// Mitsubishi GX Developer project: 壓碗機_20130207   PLC: FX1N

PROGRAM MAIN
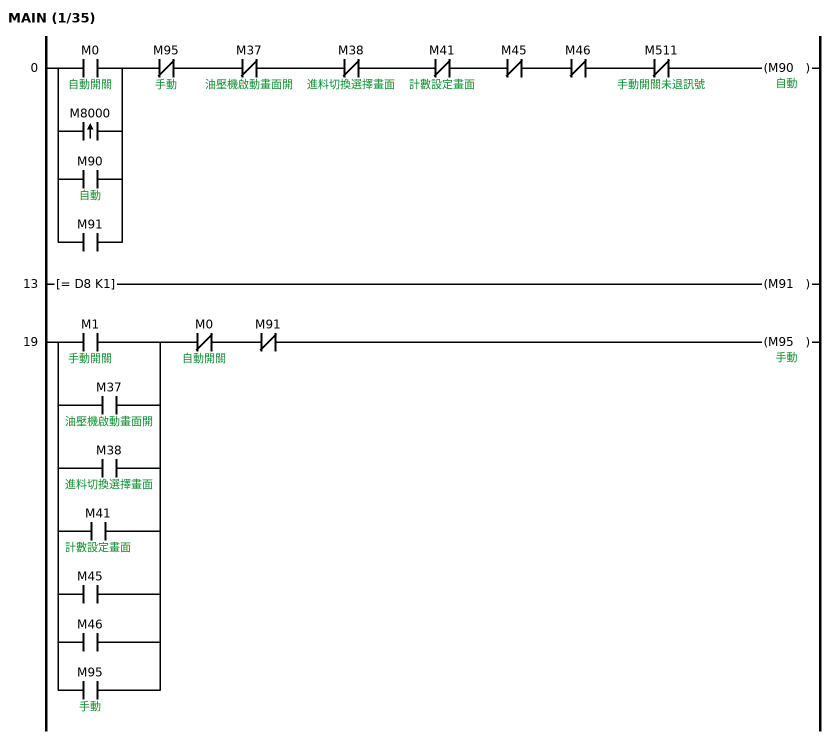
0     LD      M0  ; 自動開關
      ORP     M8000
      OR      M90  ; 自動
      OR      M91
      ANI     M95  ; 手動
      ANI     M37  ; 油壓機啟動畫面開
      ANI     M38  ; 進料切換選擇畫面
      ANI     M41  ; 計數設定畫面
      ANI     M45
      ANI     M46
      ANI     M511  ; 手動開關未退訊號
      OUT     M90  ; 自動
13    LD=     D8 K1
      OUT     M91
19    LD      M1  ; 手動開關
      OR      M37  ; 油壓機啟動畫面開
      OR      M38  ; 進料切換選擇畫面
      OR      M41  ; 計數設定畫面
      OR      M45
      OR      M46
      OR      M95  ; 手動
      ANI     M0  ; 自動開關
      ANI     M91
      OUT     M95  ; 手動
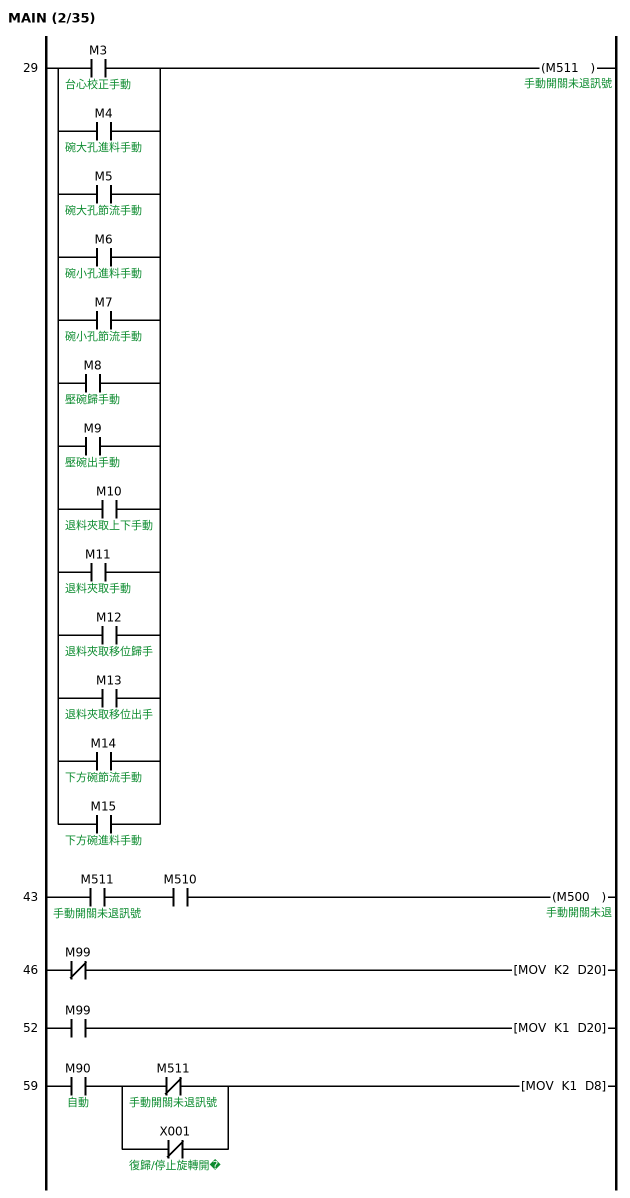
29    LD      M3  ; 台心校正手動
      OR      M4  ; 碗大孔進料手動
      OR      M5  ; 碗大孔節流手動
      OR      M6  ; 碗小孔進料手動
      OR      M7  ; 碗小孔節流手動
      OR      M8  ; 壓碗歸手動
      OR      M9  ; 壓碗出手動
      OR      M10  ; 退料夾取上下手動
      OR      M11  ; 退料夾取手動
      OR      M12  ; 退料夾取移位歸手
      OR      M13  ; 退料夾取移位出手
      OR      M14  ; 下方碗節流手動
      OR      M15  ; 下方碗進料手動
      OUT     M511  ; 手動開關未退訊號
43    LD      M511  ; 手動開關未退訊號
      AND     M510
      OUT     M500  ; 手動開關未退
46    LDI     M99
      MOV     K2 D20
52    LD      M99
      MOV     K1 D20
59    LD      M90  ; 自動
      LDI     M511  ; 手動開關未退訊號
      ORI     X001  ; 復歸/停止旋轉開�
      ANB
      MOV     K1 D8
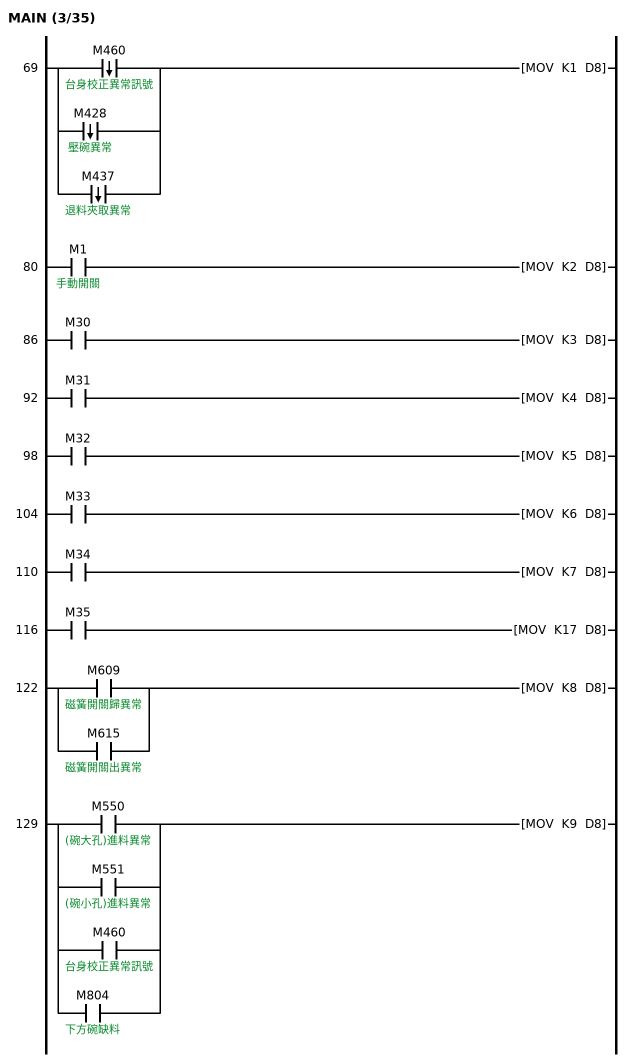
69    LDF     M460  ; 台身校正異常訊號
      ORF     M428  ; 壓碗異常
      ORF     M437  ; 退料夾取異常
      MOV     K1 D8
80    LD      M1  ; 手動開關
      MOV     K2 D8
86    LD      M30
      MOV     K3 D8
92    LD      M31
      MOV     K4 D8
98    LD      M32
      MOV     K5 D8
104   LD      M33
      MOV     K6 D8
110   LD      M34
      MOV     K7 D8
116   LD      M35
      MOV     K17 D8
122   LD      M609  ; 磁簧開關歸異常
      OR      M615  ; 磁簧開關出異常
      MOV     K8 D8
129   LD      M550  ; (碗大孔)進料異常
      OR      M551  ; (碗小孔)進料異常
      OR      M460  ; 台身校正異常訊號
      OR      M804  ; 下方碗缺料
      MOV     K9 D8
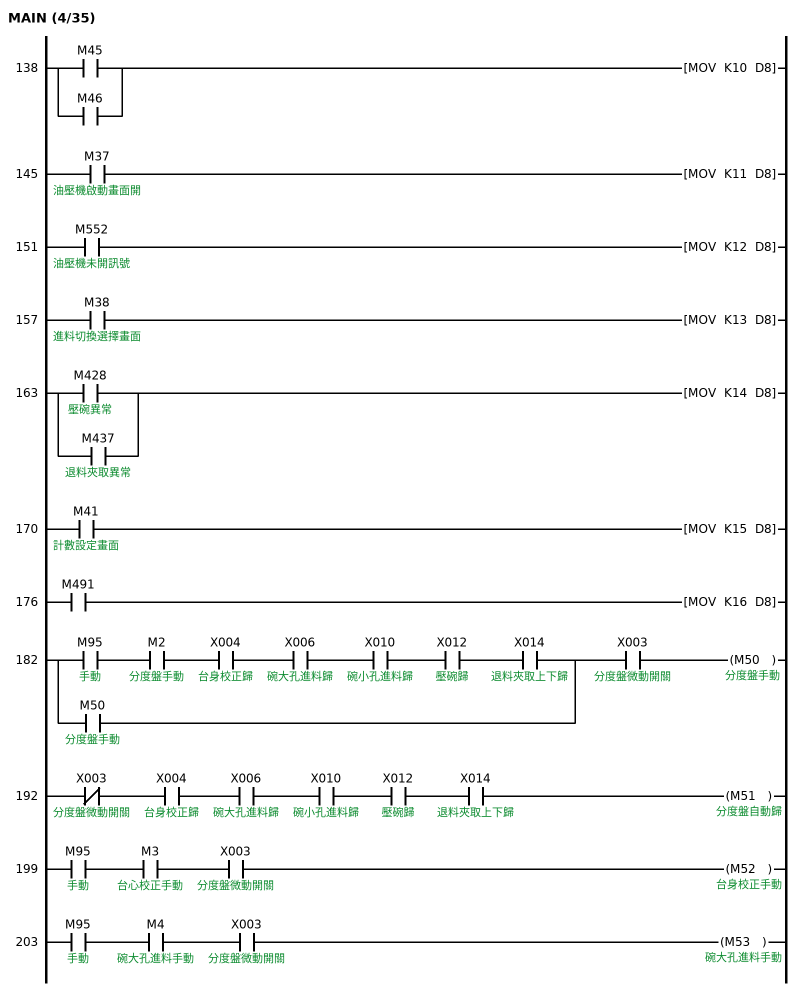
138   LD      M45
      OR      M46
      MOV     K10 D8
145   LD      M37  ; 油壓機啟動畫面開
      MOV     K11 D8
151   LD      M552  ; 油壓機未開訊號
      MOV     K12 D8
157   LD      M38  ; 進料切換選擇畫面
      MOV     K13 D8
163   LD      M428  ; 壓碗異常
      OR      M437  ; 退料夾取異常
      MOV     K14 D8
170   LD      M41  ; 計數設定畫面
      MOV     K15 D8
176   LD      M491
      MOV     K16 D8
182   LD      M95  ; 手動
      AND     M2  ; 分度盤手動
      AND     X004  ; 台身校正歸
      AND     X006  ; 碗大孔進料歸
      AND     X010  ; 碗小孔進料歸
      AND     X012  ; 壓碗歸
      AND     X014  ; 退料夾取上下歸
      OR      M50  ; 分度盤手動
      AND     X003  ; 分度盤微動開關
      OUT     M50  ; 分度盤手動
192   LDI     X003  ; 分度盤微動開關
      AND     X004  ; 台身校正歸
      AND     X006  ; 碗大孔進料歸
      AND     X010  ; 碗小孔進料歸
      AND     X012  ; 壓碗歸
      AND     X014  ; 退料夾取上下歸
      OUT     M51  ; 分度盤自動歸
199   LD      M95  ; 手動
      AND     M3  ; 台心校正手動
      AND     X003  ; 分度盤微動開關
      OUT     M52  ; 台身校正手動
203   LD      M95  ; 手動
      AND     M4  ; 碗大孔進料手動
      AND     X003  ; 分度盤微動開關
      OUT     M53  ; 碗大孔進料手動
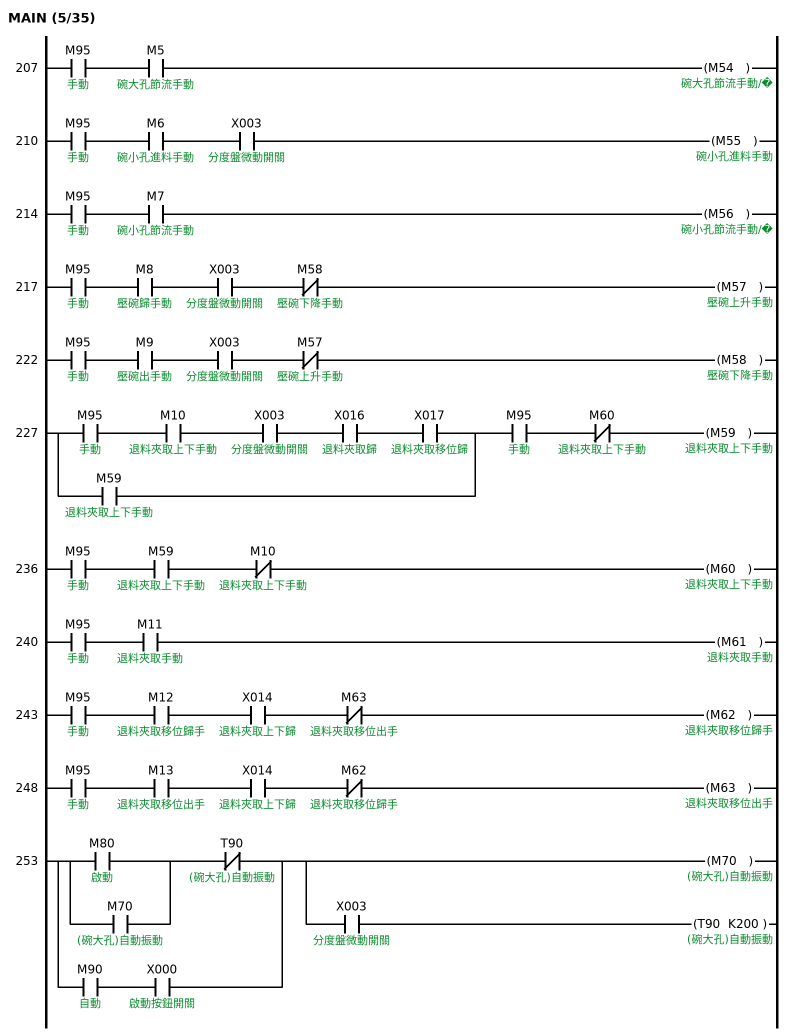
207   LD      M95  ; 手動
      AND     M5  ; 碗大孔節流手動
      OUT     M54  ; 碗大孔節流手動/�
210   LD      M95  ; 手動
      AND     M6  ; 碗小孔進料手動
      AND     X003  ; 分度盤微動開關
      OUT     M55  ; 碗小孔進料手動
214   LD      M95  ; 手動
      AND     M7  ; 碗小孔節流手動
      OUT     M56  ; 碗小孔節流手動/�
217   LD      M95  ; 手動
      AND     M8  ; 壓碗歸手動
      AND     X003  ; 分度盤微動開關
      ANI     M58  ; 壓碗下降手動
      OUT     M57  ; 壓碗上升手動
222   LD      M95  ; 手動
      AND     M9  ; 壓碗出手動
      AND     X003  ; 分度盤微動開關
      ANI     M57  ; 壓碗上升手動
      OUT     M58  ; 壓碗下降手動
227   LD      M95  ; 手動
      AND     M10  ; 退料夾取上下手動
      AND     X003  ; 分度盤微動開關
      AND     X016  ; 退料夾取歸
      AND     X017  ; 退料夾取移位歸
      OR      M59  ; 退料夾取上下手動
      AND     M95  ; 手動
      ANI     M60  ; 退料夾取上下手動
      OUT     M59  ; 退料夾取上下手動
236   LD      M95  ; 手動
      AND     M59  ; 退料夾取上下手動
      ANI     M10  ; 退料夾取上下手動
      OUT     M60  ; 退料夾取上下手動
240   LD      M95  ; 手動
      AND     M11  ; 退料夾取手動
      OUT     M61  ; 退料夾取手動
243   LD      M95  ; 手動
      AND     M12  ; 退料夾取移位歸手
      AND     X014  ; 退料夾取上下歸
      ANI     M63  ; 退料夾取移位出手
      OUT     M62  ; 退料夾取移位歸手
248   LD      M95  ; 手動
      AND     M13  ; 退料夾取移位出手
      AND     X014  ; 退料夾取上下歸
      ANI     M62  ; 退料夾取移位歸手
      OUT     M63  ; 退料夾取移位出手
253   LD      M80  ; 啟動
      OR      M70  ; (碗大孔)自動振動
      ANI     T90  ; (碗大孔)自動振動
      LD      M90  ; 自動
      AND     X000  ; 啟動按鈕開關
      ORB
      OUT     M70  ; (碗大孔)自動振動
      AND     X003  ; 分度盤微動開關
      OUT     T90 K200  ; (碗大孔)自動振動
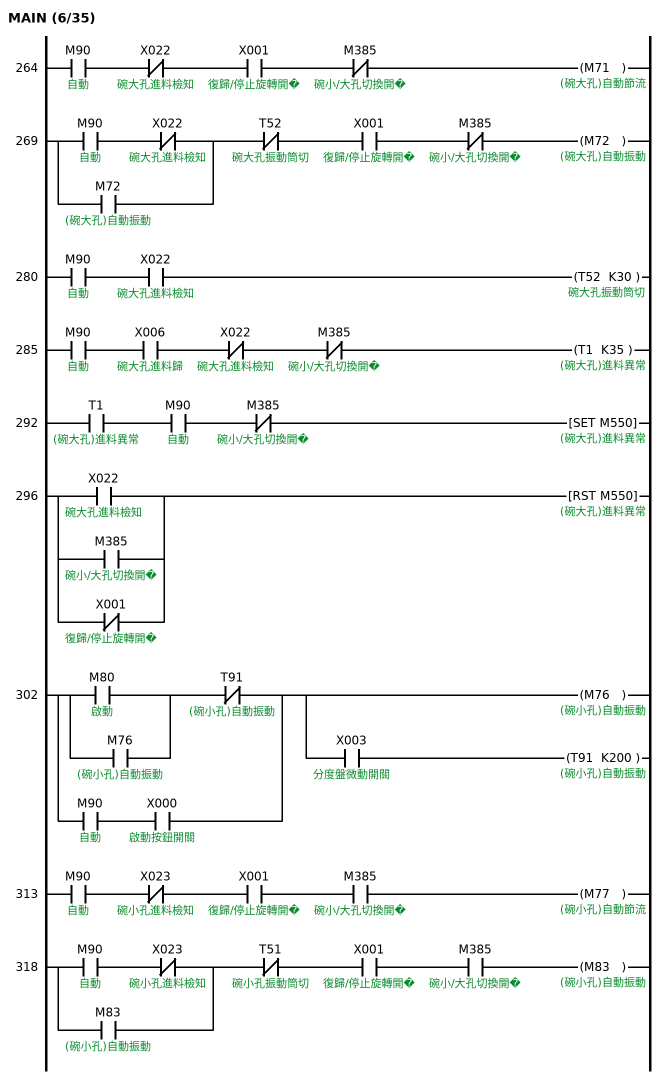
264   LD      M90  ; 自動
      ANI     X022  ; 碗大孔進料檢知
      AND     X001  ; 復歸/停止旋轉開�
      ANI     M385  ; 碗小/大孔切換開�
      OUT     M71  ; (碗大孔)自動節流
269   LD      M90  ; 自動
      ANI     X022  ; 碗大孔進料檢知
      OR      M72  ; (碗大孔)自動振動
      ANI     T52  ; 碗大孔振動筒切
      AND     X001  ; 復歸/停止旋轉開�
      ANI     M385  ; 碗小/大孔切換開�
      OUT     M72  ; (碗大孔)自動振動
280   LD      M90  ; 自動
      AND     X022  ; 碗大孔進料檢知
      OUT     T52 K30  ; 碗大孔振動筒切
285   LD      M90  ; 自動
      AND     X006  ; 碗大孔進料歸
      ANI     X022  ; 碗大孔進料檢知
      ANI     M385  ; 碗小/大孔切換開�
      OUT     T1 K35  ; (碗大孔)進料異常
292   LD      T1  ; (碗大孔)進料異常
      AND     M90  ; 自動
      ANI     M385  ; 碗小/大孔切換開�
      SET     M550  ; (碗大孔)進料異常
296   LD      X022  ; 碗大孔進料檢知
      OR      M385  ; 碗小/大孔切換開�
      ORI     X001  ; 復歸/停止旋轉開�
      RST     M550  ; (碗大孔)進料異常
302   LD      M80  ; 啟動
      OR      M76  ; (碗小孔)自動振動
      ANI     T91  ; (碗小孔)自動振動
      LD      M90  ; 自動
      AND     X000  ; 啟動按鈕開關
      ORB
      OUT     M76  ; (碗小孔)自動振動
      AND     X003  ; 分度盤微動開關
      OUT     T91 K200  ; (碗小孔)自動振動
313   LD      M90  ; 自動
      ANI     X023  ; 碗小孔進料檢知
      AND     X001  ; 復歸/停止旋轉開�
      AND     M385  ; 碗小/大孔切換開�
      OUT     M77  ; (碗小孔)自動節流
318   LD      M90  ; 自動
      ANI     X023  ; 碗小孔進料檢知
      OR      M83  ; (碗小孔)自動振動
      ANI     T51  ; 碗小孔振動筒切
      AND     X001  ; 復歸/停止旋轉開�
      AND     M385  ; 碗小/大孔切換開�
      OUT     M83  ; (碗小孔)自動振動
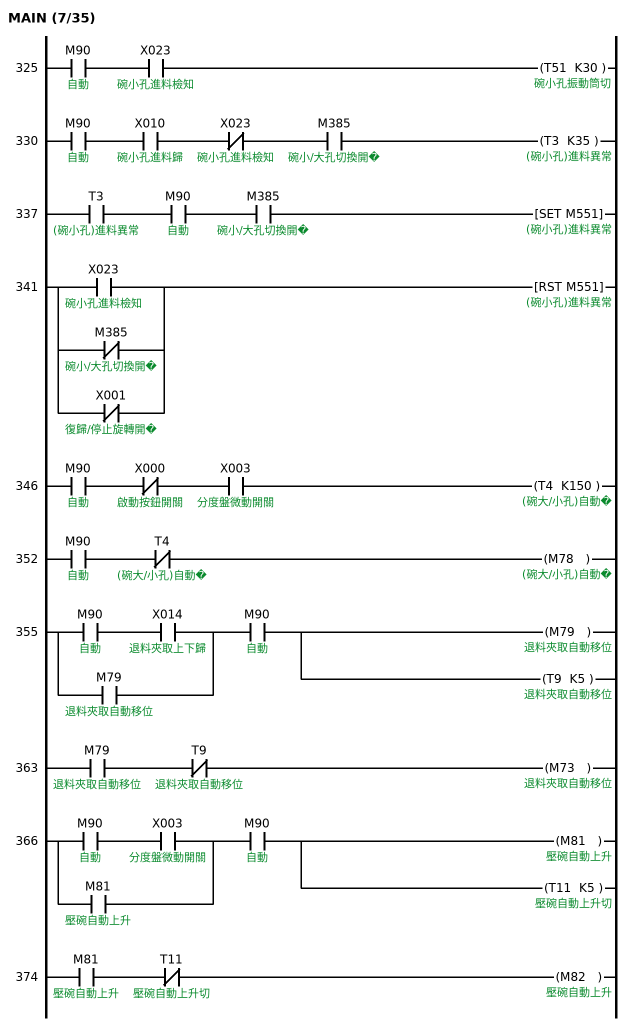
325   LD      M90  ; 自動
      AND     X023  ; 碗小孔進料檢知
      OUT     T51 K30  ; 碗小孔振動筒切
330   LD      M90  ; 自動
      AND     X010  ; 碗小孔進料歸
      ANI     X023  ; 碗小孔進料檢知
      AND     M385  ; 碗小/大孔切換開�
      OUT     T3 K35  ; (碗小孔)進料異常
337   LD      T3  ; (碗小孔)進料異常
      AND     M90  ; 自動
      AND     M385  ; 碗小/大孔切換開�
      SET     M551  ; (碗小孔)進料異常
341   LD      X023  ; 碗小孔進料檢知
      ORI     M385  ; 碗小/大孔切換開�
      ORI     X001  ; 復歸/停止旋轉開�
      RST     M551  ; (碗小孔)進料異常
346   LD      M90  ; 自動
      ANI     X000  ; 啟動按鈕開關
      AND     X003  ; 分度盤微動開關
      OUT     T4 K150  ; (碗大/小孔)自動�
352   LD      M90  ; 自動
      ANI     T4  ; (碗大/小孔)自動�
      OUT     M78  ; (碗大/小孔)自動�
355   LD      M90  ; 自動
      AND     X014  ; 退料夾取上下歸
      OR      M79  ; 退料夾取自動移位
      AND     M90  ; 自動
      OUT     M79  ; 退料夾取自動移位
      OUT     T9 K5  ; 退料夾取自動移位
363   LD      M79  ; 退料夾取自動移位
      ANI     T9  ; 退料夾取自動移位
      OUT     M73  ; 退料夾取自動移位
366   LD      M90  ; 自動
      AND     X003  ; 分度盤微動開關
      OR      M81  ; 壓碗自動上升
      AND     M90  ; 自動
      OUT     M81  ; 壓碗自動上升
      OUT     T11 K5  ; 壓碗自動上升切
374   LD      M81  ; 壓碗自動上升
      ANI     T11  ; 壓碗自動上升切
      OUT     M82  ; 壓碗自動上升
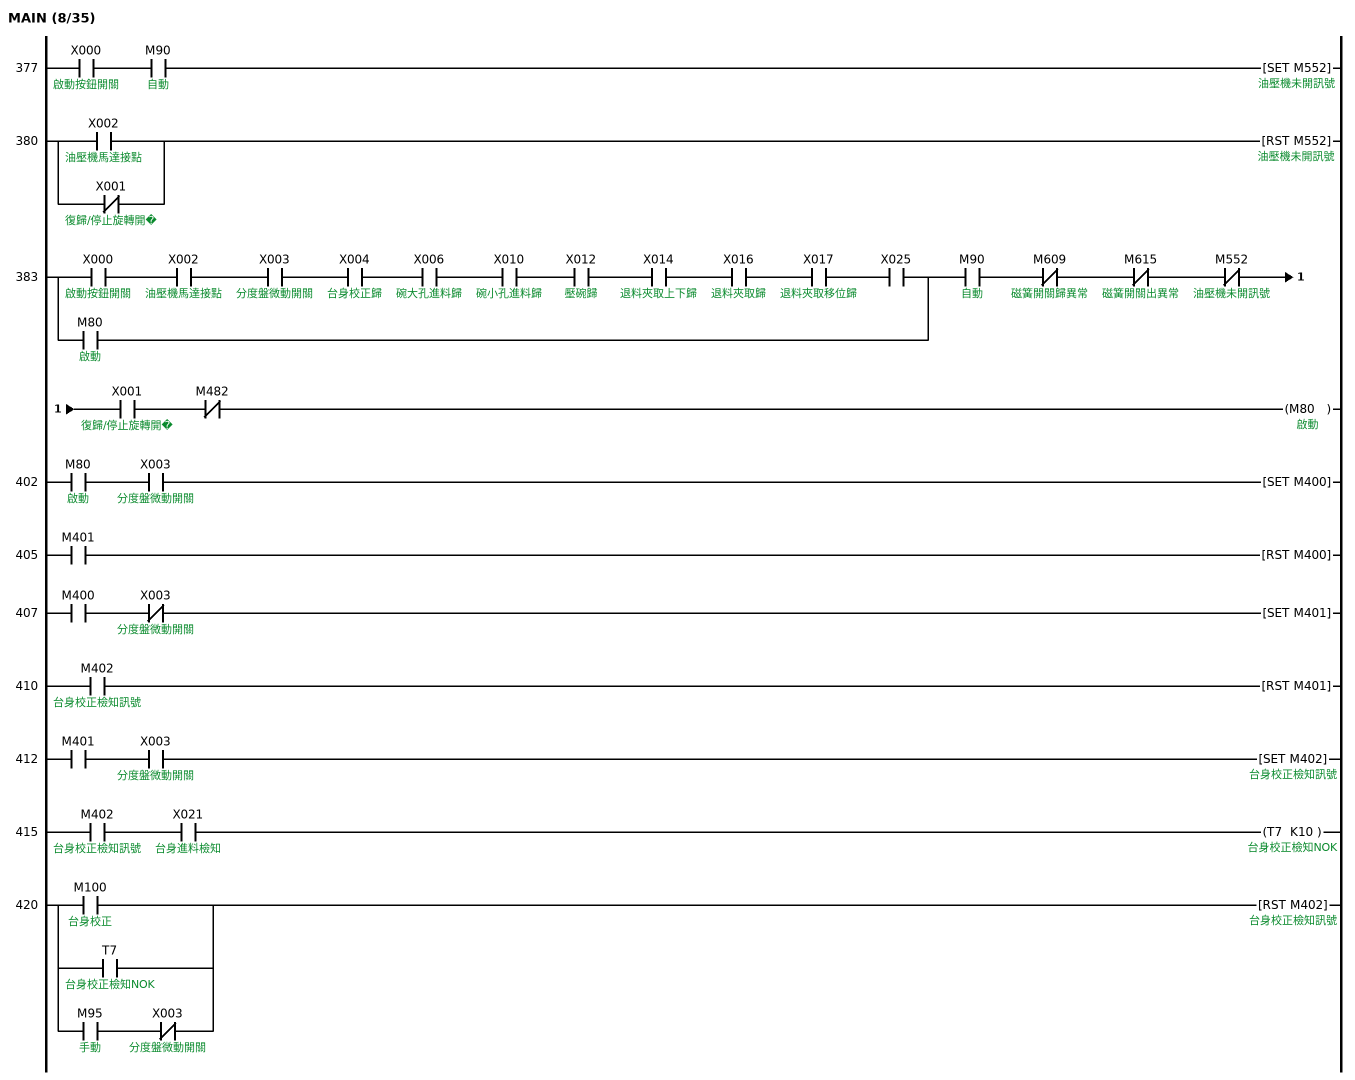
377   LD      X000  ; 啟動按鈕開關
      AND     M90  ; 自動
      SET     M552  ; 油壓機未開訊號
380   LD      X002  ; 油壓機馬達接點
      ORI     X001  ; 復歸/停止旋轉開�
      RST     M552  ; 油壓機未開訊號
383   LD      X000  ; 啟動按鈕開關
      AND     X002  ; 油壓機馬達接點
      AND     X003  ; 分度盤微動開關
      AND     X004  ; 台身校正歸
      AND     X006  ; 碗大孔進料歸
      AND     X010  ; 碗小孔進料歸
      AND     X012  ; 壓碗歸
      AND     X014  ; 退料夾取上下歸
      AND     X016  ; 退料夾取歸
      AND     X017  ; 退料夾取移位歸
      AND     X025
      OR      M80  ; 啟動
      AND     M90  ; 自動
      ANI     M609  ; 磁簧開關歸異常
      ANI     M615  ; 磁簧開關出異常
      ANI     M552  ; 油壓機未開訊號
      AND     X001  ; 復歸/停止旋轉開�
      ANI     M482
      OUT     M80  ; 啟動
402   LD      M80  ; 啟動
      AND     X003  ; 分度盤微動開關
      SET     M400
405   LD      M401
      RST     M400
407   LD      M400
      ANI     X003  ; 分度盤微動開關
      SET     M401
410   LD      M402  ; 台身校正檢知訊號
      RST     M401
412   LD      M401
      AND     X003  ; 分度盤微動開關
      SET     M402  ; 台身校正檢知訊號
415   LD      M402  ; 台身校正檢知訊號
      AND     X021  ; 台身進料檢知
      OUT     T7 K10  ; 台身校正檢知NOK
420   LD      M100  ; 台身校正
      OR      T7  ; 台身校正檢知NOK
      LD      M95  ; 手動
      ANI     X003  ; 分度盤微動開關
      ORB
      RST     M402  ; 台身校正檢知訊號
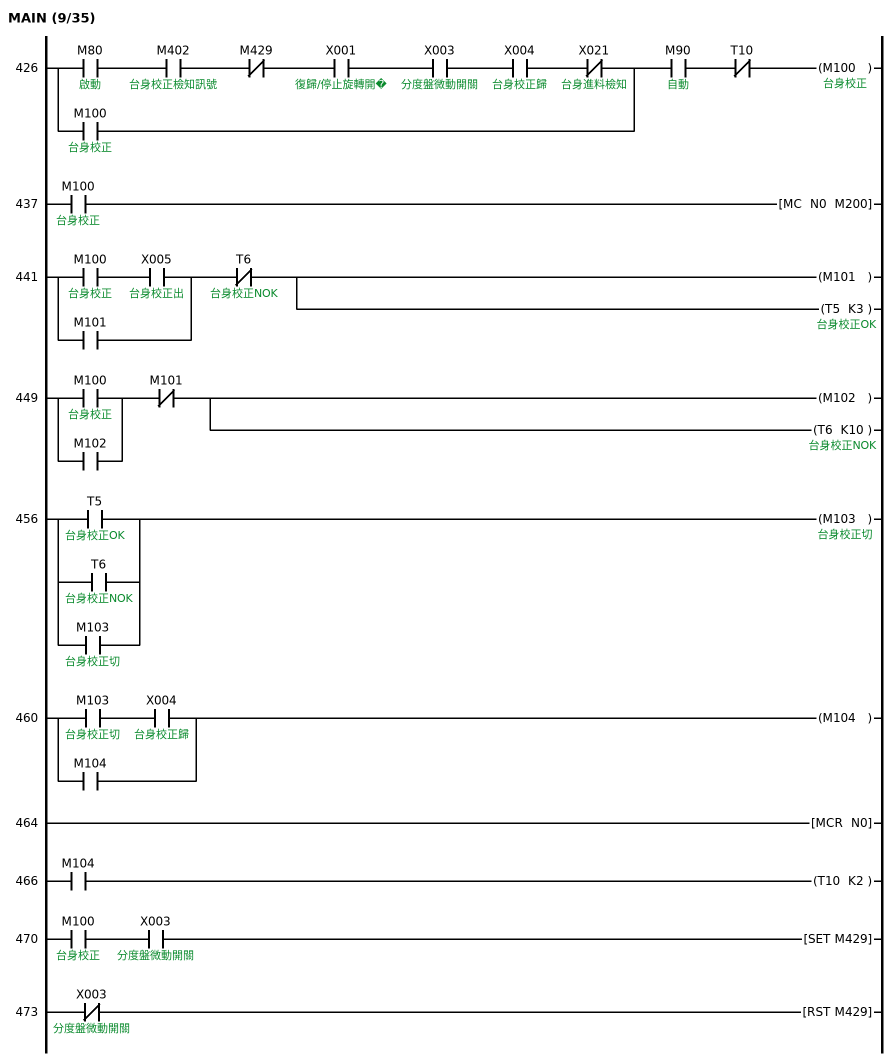
426   LD      M80  ; 啟動
      AND     M402  ; 台身校正檢知訊號
      ANI     M429
      AND     X001  ; 復歸/停止旋轉開�
      AND     X003  ; 分度盤微動開關
      AND     X004  ; 台身校正歸
      ANI     X021  ; 台身進料檢知
      OR      M100  ; 台身校正
      AND     M90  ; 自動
      ANI     T10
      OUT     M100  ; 台身校正
437   LD      M100  ; 台身校正
      MC      N0 M200
441   LD      M100  ; 台身校正
      AND     X005  ; 台身校正出
      OR      M101
      ANI     T6  ; 台身校正NOK
      OUT     M101
      OUT     T5 K3  ; 台身校正OK
449   LD      M100  ; 台身校正
      OR      M102
      ANI     M101
      OUT     M102
      OUT     T6 K10  ; 台身校正NOK
456   LD      T5  ; 台身校正OK
      OR      T6  ; 台身校正NOK
      OR      M103  ; 台身校正切
      OUT     M103  ; 台身校正切
460   LD      M103  ; 台身校正切
      AND     X004  ; 台身校正歸
      OR      M104
      OUT     M104
464   MCR     N0
466   LD      M104
      OUT     T10 K2
470   LD      M100  ; 台身校正
      AND     X003  ; 分度盤微動開關
      SET     M429
473   LDI     X003  ; 分度盤微動開關
      RST     M429
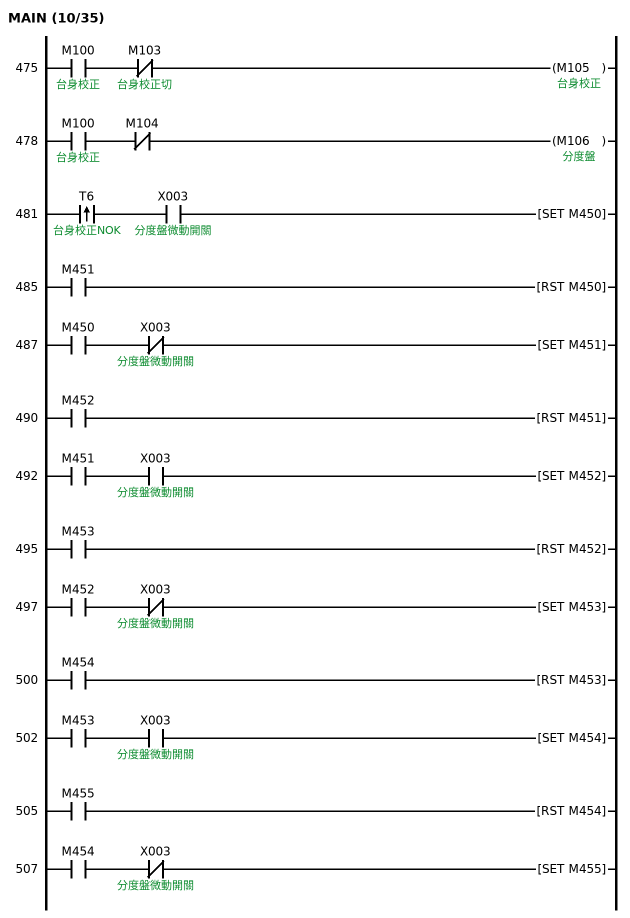
475   LD      M100  ; 台身校正
      ANI     M103  ; 台身校正切
      OUT     M105  ; 台身校正
478   LD      M100  ; 台身校正
      ANI     M104
      OUT     M106  ; 分度盤
481   LDP     T6  ; 台身校正NOK
      AND     X003  ; 分度盤微動開關
      SET     M450
485   LD      M451
      RST     M450
487   LD      M450
      ANI     X003  ; 分度盤微動開關
      SET     M451
490   LD      M452
      RST     M451
492   LD      M451
      AND     X003  ; 分度盤微動開關
      SET     M452
495   LD      M453
      RST     M452
497   LD      M452
      ANI     X003  ; 分度盤微動開關
      SET     M453
500   LD      M454
      RST     M453
502   LD      M453
      AND     X003  ; 分度盤微動開關
      SET     M454
505   LD      M455
      RST     M454
507   LD      M454
      ANI     X003  ; 分度盤微動開關
      SET     M455
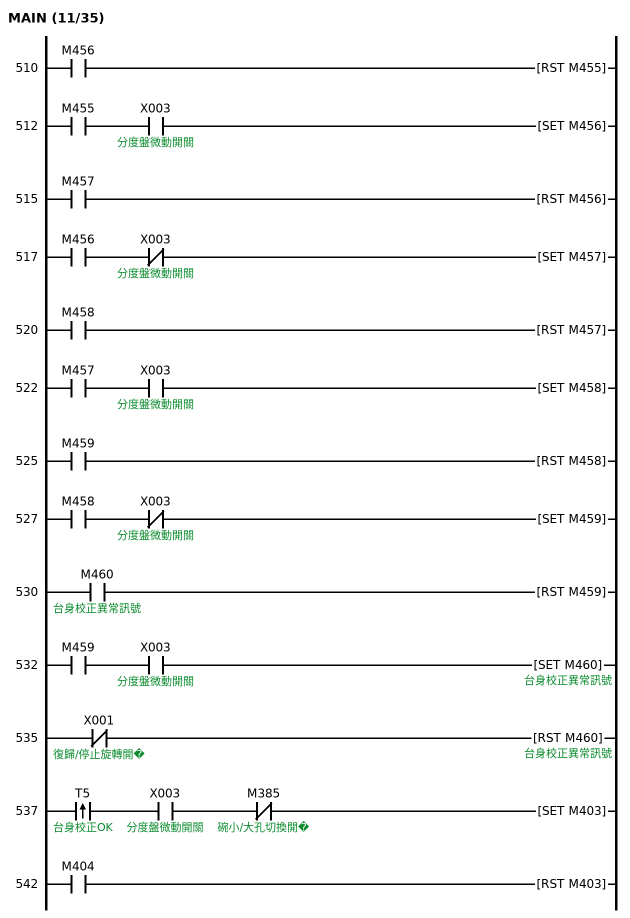
510   LD      M456
      RST     M455
512   LD      M455
      AND     X003  ; 分度盤微動開關
      SET     M456
515   LD      M457
      RST     M456
517   LD      M456
      ANI     X003  ; 分度盤微動開關
      SET     M457
520   LD      M458
      RST     M457
522   LD      M457
      AND     X003  ; 分度盤微動開關
      SET     M458
525   LD      M459
      RST     M458
527   LD      M458
      ANI     X003  ; 分度盤微動開關
      SET     M459
530   LD      M460  ; 台身校正異常訊號
      RST     M459
532   LD      M459
      AND     X003  ; 分度盤微動開關
      SET     M460  ; 台身校正異常訊號
535   LDI     X001  ; 復歸/停止旋轉開�
      RST     M460  ; 台身校正異常訊號
537   LDP     T5  ; 台身校正OK
      AND     X003  ; 分度盤微動開關
      ANI     M385  ; 碗小/大孔切換開�
      SET     M403
542   LD      M404
      RST     M403
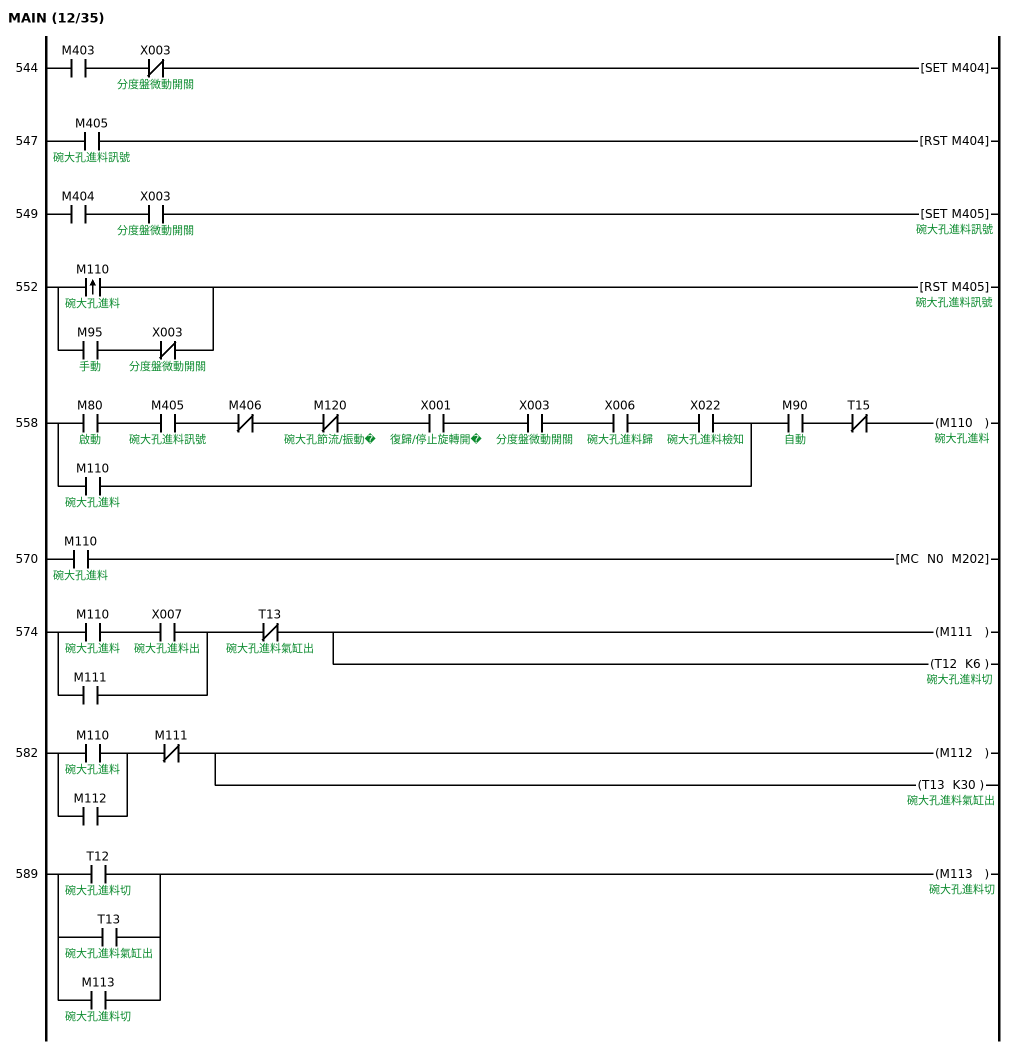
544   LD      M403
      ANI     X003  ; 分度盤微動開關
      SET     M404
547   LD      M405  ; 碗大孔進料訊號
      RST     M404
549   LD      M404
      AND     X003  ; 分度盤微動開關
      SET     M405  ; 碗大孔進料訊號
552   LDP     M110  ; 碗大孔進料
      LD      M95  ; 手動
      ANI     X003  ; 分度盤微動開關
      ORB
      RST     M405  ; 碗大孔進料訊號
558   LD      M80  ; 啟動
      AND     M405  ; 碗大孔進料訊號
      ANI     M406
      ANI     M120  ; 碗大孔節流/振動�
      AND     X001  ; 復歸/停止旋轉開�
      AND     X003  ; 分度盤微動開關
      AND     X006  ; 碗大孔進料歸
      AND     X022  ; 碗大孔進料檢知
      OR      M110  ; 碗大孔進料
      AND     M90  ; 自動
      ANI     T15
      OUT     M110  ; 碗大孔進料
570   LD      M110  ; 碗大孔進料
      MC      N0 M202
574   LD      M110  ; 碗大孔進料
      AND     X007  ; 碗大孔進料出
      OR      M111
      ANI     T13  ; 碗大孔進料氣缸出
      OUT     M111
      OUT     T12 K6  ; 碗大孔進料切
582   LD      M110  ; 碗大孔進料
      OR      M112
      ANI     M111
      OUT     M112
      OUT     T13 K30  ; 碗大孔進料氣缸出
589   LD      T12  ; 碗大孔進料切
      OR      T13  ; 碗大孔進料氣缸出
      OR      M113  ; 碗大孔進料切
      OUT     M113  ; 碗大孔進料切
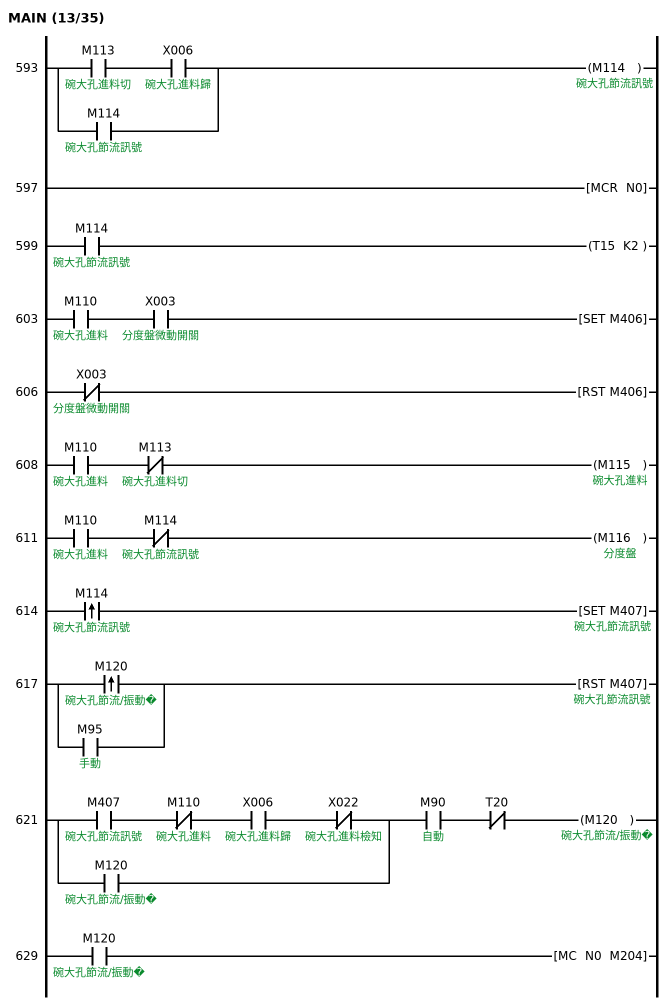
593   LD      M113  ; 碗大孔進料切
      AND     X006  ; 碗大孔進料歸
      OR      M114  ; 碗大孔節流訊號
      OUT     M114  ; 碗大孔節流訊號
597   MCR     N0
599   LD      M114  ; 碗大孔節流訊號
      OUT     T15 K2
603   LD      M110  ; 碗大孔進料
      AND     X003  ; 分度盤微動開關
      SET     M406
606   LDI     X003  ; 分度盤微動開關
      RST     M406
608   LD      M110  ; 碗大孔進料
      ANI     M113  ; 碗大孔進料切
      OUT     M115  ; 碗大孔進料
611   LD      M110  ; 碗大孔進料
      ANI     M114  ; 碗大孔節流訊號
      OUT     M116  ; 分度盤
614   LDP     M114  ; 碗大孔節流訊號
      SET     M407  ; 碗大孔節流訊號
617   LDP     M120  ; 碗大孔節流/振動�
      OR      M95  ; 手動
      RST     M407  ; 碗大孔節流訊號
621   LD      M407  ; 碗大孔節流訊號
      ANI     M110  ; 碗大孔進料
      AND     X006  ; 碗大孔進料歸
      ANI     X022  ; 碗大孔進料檢知
      OR      M120  ; 碗大孔節流/振動�
      AND     M90  ; 自動
      ANI     T20
      OUT     M120  ; 碗大孔節流/振動�
629   LD      M120  ; 碗大孔節流/振動�
      MC      N0 M204
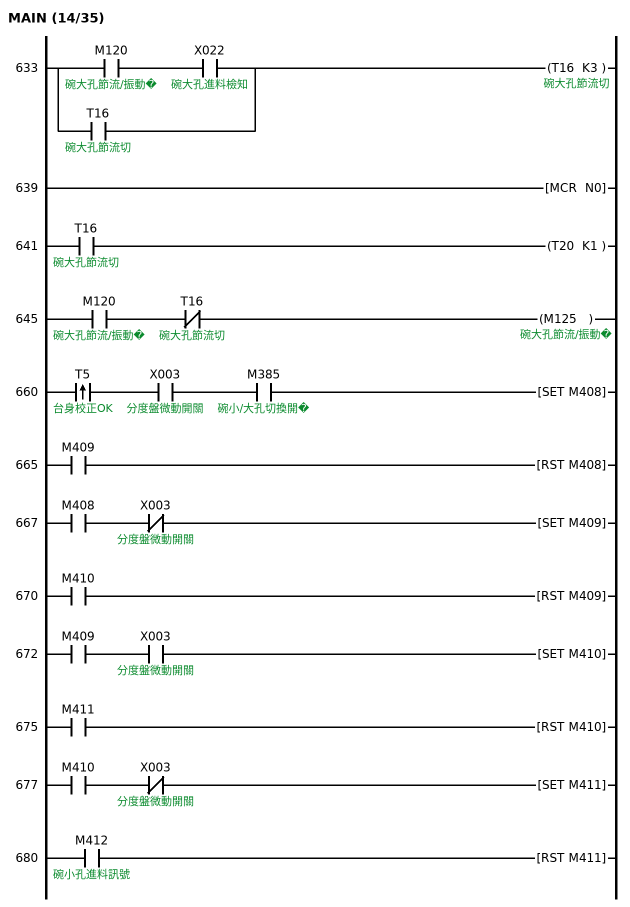
633   LD      M120  ; 碗大孔節流/振動�
      AND     X022  ; 碗大孔進料檢知
      OR      T16  ; 碗大孔節流切
      OUT     T16 K3  ; 碗大孔節流切
639   MCR     N0
641   LD      T16  ; 碗大孔節流切
      OUT     T20 K1
645   LD      M120  ; 碗大孔節流/振動�
      ANI     T16  ; 碗大孔節流切
      OUT     M125  ; 碗大孔節流/振動�
660   LDP     T5  ; 台身校正OK
      AND     X003  ; 分度盤微動開關
      AND     M385  ; 碗小/大孔切換開�
      SET     M408
665   LD      M409
      RST     M408
667   LD      M408
      ANI     X003  ; 分度盤微動開關
      SET     M409
670   LD      M410
      RST     M409
672   LD      M409
      AND     X003  ; 分度盤微動開關
      SET     M410
675   LD      M411
      RST     M410
677   LD      M410
      ANI     X003  ; 分度盤微動開關
      SET     M411
680   LD      M412  ; 碗小孔進料訊號
      RST     M411
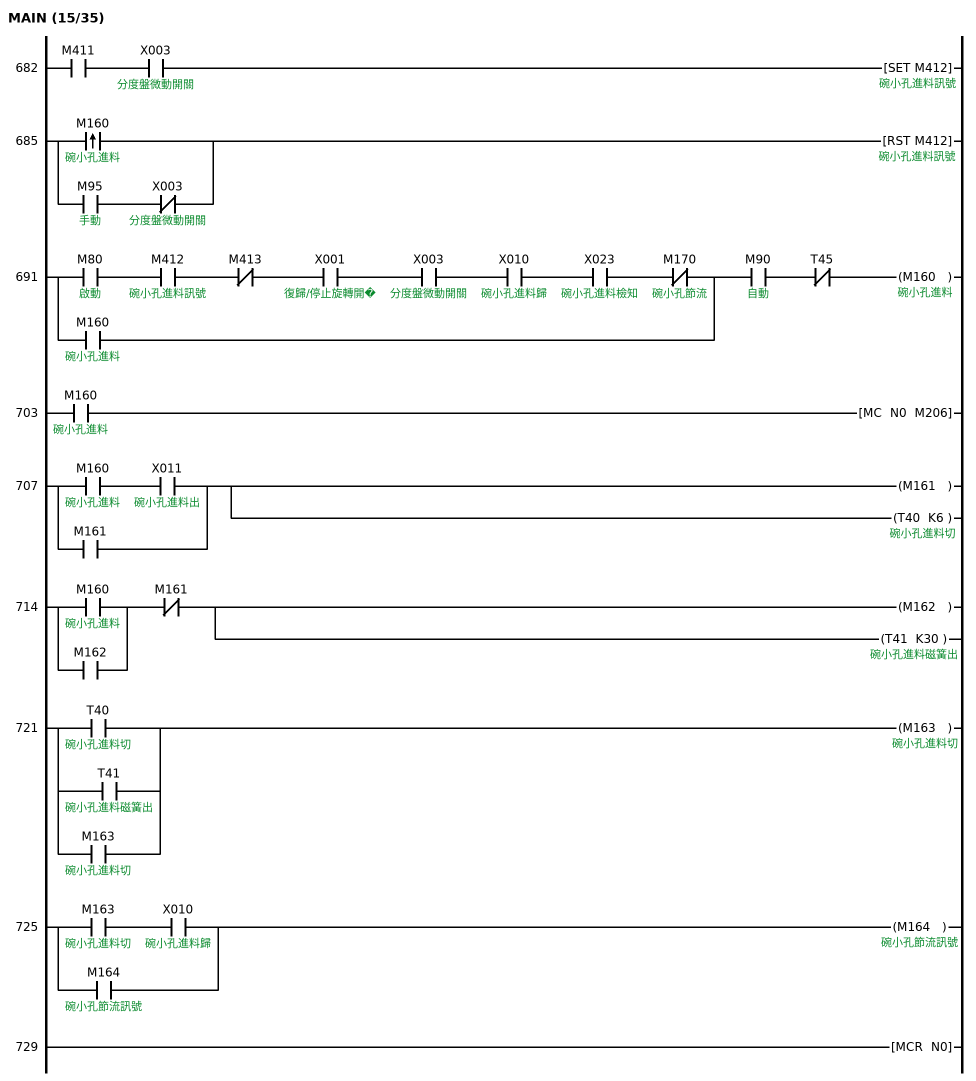
682   LD      M411
      AND     X003  ; 分度盤微動開關
      SET     M412  ; 碗小孔進料訊號
685   LDP     M160  ; 碗小孔進料
      LD      M95  ; 手動
      ANI     X003  ; 分度盤微動開關
      ORB
      RST     M412  ; 碗小孔進料訊號
691   LD      M80  ; 啟動
      AND     M412  ; 碗小孔進料訊號
      ANI     M413
      AND     X001  ; 復歸/停止旋轉開�
      AND     X003  ; 分度盤微動開關
      AND     X010  ; 碗小孔進料歸
      AND     X023  ; 碗小孔進料檢知
      ANI     M170  ; 碗小孔節流
      OR      M160  ; 碗小孔進料
      AND     M90  ; 自動
      ANI     T45
      OUT     M160  ; 碗小孔進料
703   LD      M160  ; 碗小孔進料
      MC      N0 M206
707   LD      M160  ; 碗小孔進料
      AND     X011  ; 碗小孔進料出
      OR      M161
      OUT     M161
      OUT     T40 K6  ; 碗小孔進料切
714   LD      M160  ; 碗小孔進料
      OR      M162
      ANI     M161
      OUT     M162
      OUT     T41 K30  ; 碗小孔進料磁簧出
721   LD      T40  ; 碗小孔進料切
      OR      T41  ; 碗小孔進料磁簧出
      OR      M163  ; 碗小孔進料切
      OUT     M163  ; 碗小孔進料切
725   LD      M163  ; 碗小孔進料切
      AND     X010  ; 碗小孔進料歸
      OR      M164  ; 碗小孔節流訊號
      OUT     M164  ; 碗小孔節流訊號
729   MCR     N0
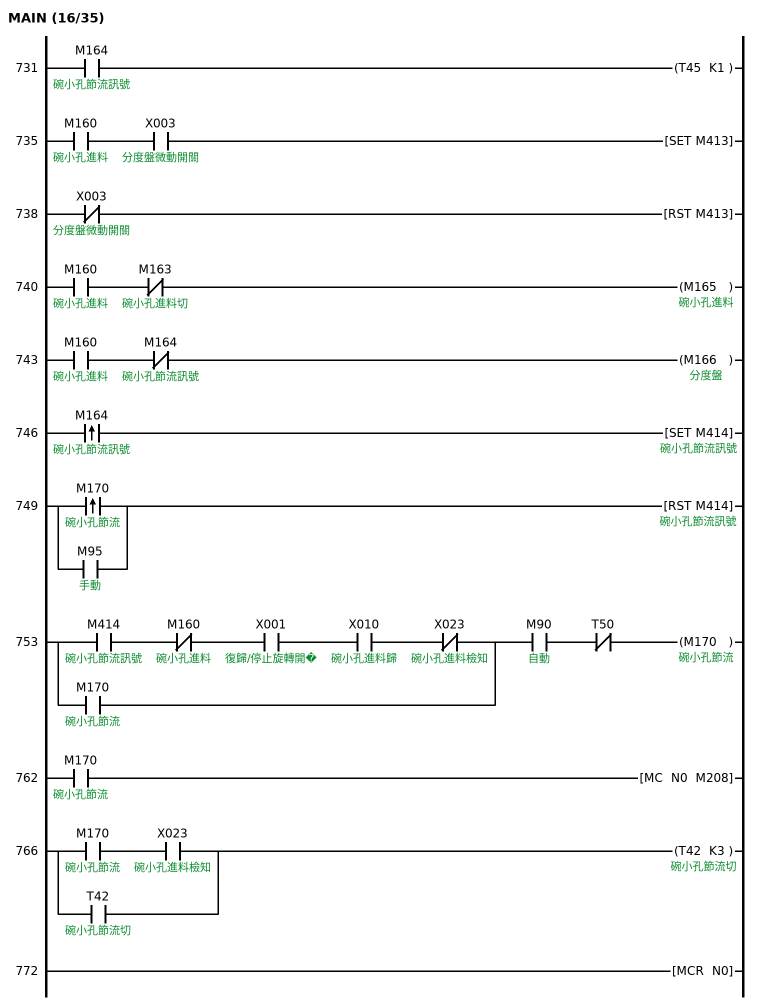
731   LD      M164  ; 碗小孔節流訊號
      OUT     T45 K1
735   LD      M160  ; 碗小孔進料
      AND     X003  ; 分度盤微動開關
      SET     M413
738   LDI     X003  ; 分度盤微動開關
      RST     M413
740   LD      M160  ; 碗小孔進料
      ANI     M163  ; 碗小孔進料切
      OUT     M165  ; 碗小孔進料
743   LD      M160  ; 碗小孔進料
      ANI     M164  ; 碗小孔節流訊號
      OUT     M166  ; 分度盤
746   LDP     M164  ; 碗小孔節流訊號
      SET     M414  ; 碗小孔節流訊號
749   LDP     M170  ; 碗小孔節流
      OR      M95  ; 手動
      RST     M414  ; 碗小孔節流訊號
753   LD      M414  ; 碗小孔節流訊號
      ANI     M160  ; 碗小孔進料
      AND     X001  ; 復歸/停止旋轉開�
      AND     X010  ; 碗小孔進料歸
      ANI     X023  ; 碗小孔進料檢知
      OR      M170  ; 碗小孔節流
      AND     M90  ; 自動
      ANI     T50
      OUT     M170  ; 碗小孔節流
762   LD      M170  ; 碗小孔節流
      MC      N0 M208
766   LD      M170  ; 碗小孔節流
      AND     X023  ; 碗小孔進料檢知
      OR      T42  ; 碗小孔節流切
      OUT     T42 K3  ; 碗小孔節流切
772   MCR     N0
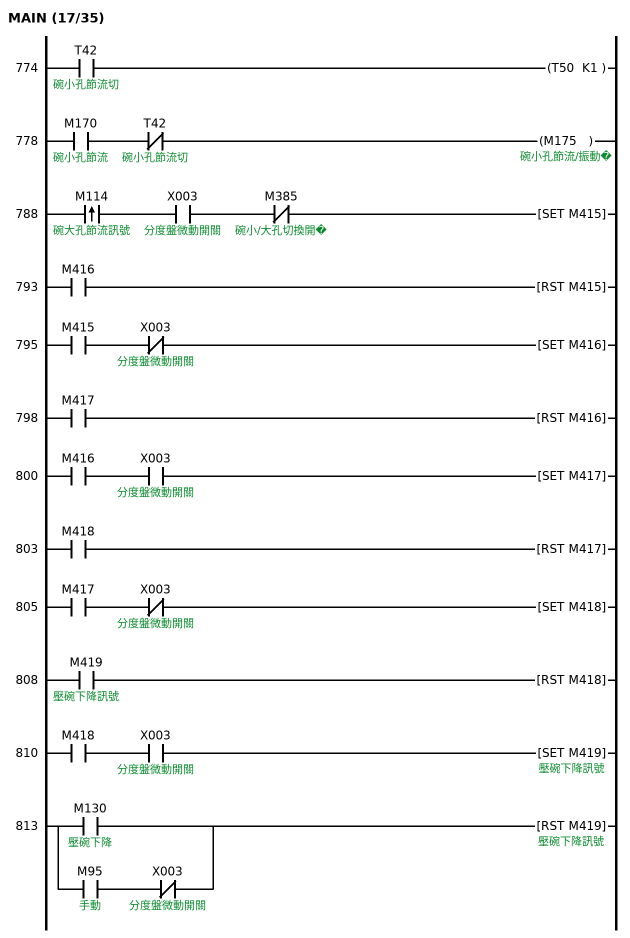
774   LD      T42  ; 碗小孔節流切
      OUT     T50 K1
778   LD      M170  ; 碗小孔節流
      ANI     T42  ; 碗小孔節流切
      OUT     M175  ; 碗小孔節流/振動�
788   LDP     M114  ; 碗大孔節流訊號
      AND     X003  ; 分度盤微動開關
      ANI     M385  ; 碗小/大孔切換開�
      SET     M415
793   LD      M416
      RST     M415
795   LD      M415
      ANI     X003  ; 分度盤微動開關
      SET     M416
798   LD      M417
      RST     M416
800   LD      M416
      AND     X003  ; 分度盤微動開關
      SET     M417
803   LD      M418
      RST     M417
805   LD      M417
      ANI     X003  ; 分度盤微動開關
      SET     M418
808   LD      M419  ; 壓碗下降訊號
      RST     M418
810   LD      M418
      AND     X003  ; 分度盤微動開關
      SET     M419  ; 壓碗下降訊號
813   LD      M130  ; 壓碗下降
      LD      M95  ; 手動
      ANI     X003  ; 分度盤微動開關
      ORB
      RST     M419  ; 壓碗下降訊號
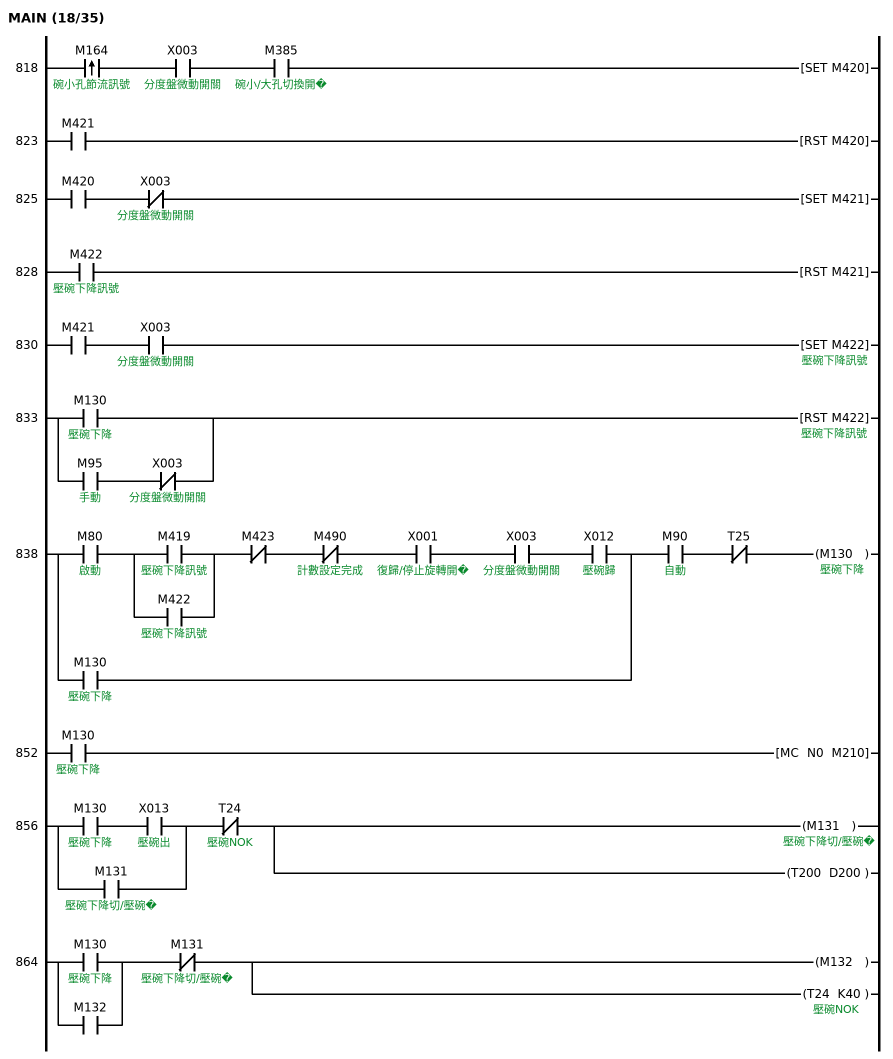
818   LDP     M164  ; 碗小孔節流訊號
      AND     X003  ; 分度盤微動開關
      AND     M385  ; 碗小/大孔切換開�
      SET     M420
823   LD      M421
      RST     M420
825   LD      M420
      ANI     X003  ; 分度盤微動開關
      SET     M421
828   LD      M422  ; 壓碗下降訊號
      RST     M421
830   LD      M421
      AND     X003  ; 分度盤微動開關
      SET     M422  ; 壓碗下降訊號
833   LD      M130  ; 壓碗下降
      LD      M95  ; 手動
      ANI     X003  ; 分度盤微動開關
      ORB
      RST     M422  ; 壓碗下降訊號
838   LD      M80  ; 啟動
      LD      M419  ; 壓碗下降訊號
      OR      M422  ; 壓碗下降訊號
      ANB
      ANI     M423
      ANI     M490  ; 計數設定完成
      AND     X001  ; 復歸/停止旋轉開�
      AND     X003  ; 分度盤微動開關
      AND     X012  ; 壓碗歸
      OR      M130  ; 壓碗下降
      AND     M90  ; 自動
      ANI     T25
      OUT     M130  ; 壓碗下降
852   LD      M130  ; 壓碗下降
      MC      N0 M210
856   LD      M130  ; 壓碗下降
      AND     X013  ; 壓碗出
      OR      M131  ; 壓碗下降切/壓碗�
      ANI     T24  ; 壓碗NOK
      OUT     M131  ; 壓碗下降切/壓碗�
      OUT     T200 D200
864   LD      M130  ; 壓碗下降
      OR      M132
      ANI     M131  ; 壓碗下降切/壓碗�
      OUT     M132
      OUT     T24 K40  ; 壓碗NOK
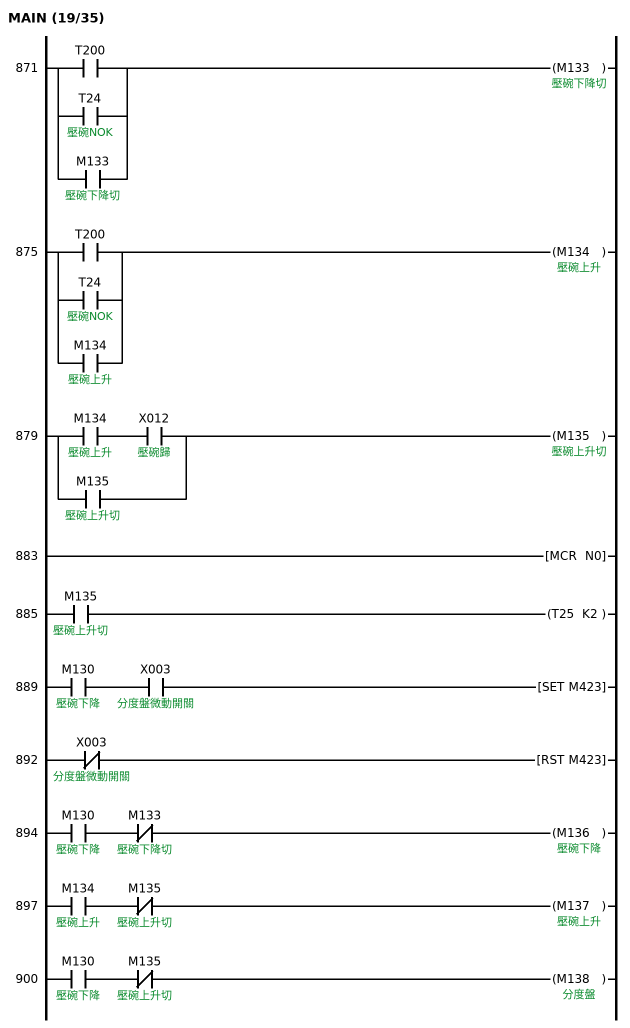
871   LD      T200
      OR      T24  ; 壓碗NOK
      OR      M133  ; 壓碗下降切
      OUT     M133  ; 壓碗下降切
875   LD      T200
      OR      T24  ; 壓碗NOK
      OR      M134  ; 壓碗上升
      OUT     M134  ; 壓碗上升
879   LD      M134  ; 壓碗上升
      AND     X012  ; 壓碗歸
      OR      M135  ; 壓碗上升切
      OUT     M135  ; 壓碗上升切
883   MCR     N0
885   LD      M135  ; 壓碗上升切
      OUT     T25 K2
889   LD      M130  ; 壓碗下降
      AND     X003  ; 分度盤微動開關
      SET     M423
892   LDI     X003  ; 分度盤微動開關
      RST     M423
894   LD      M130  ; 壓碗下降
      ANI     M133  ; 壓碗下降切
      OUT     M136  ; 壓碗下降
897   LD      M134  ; 壓碗上升
      ANI     M135  ; 壓碗上升切
      OUT     M137  ; 壓碗上升
900   LD      M130  ; 壓碗下降
      ANI     M135  ; 壓碗上升切
      OUT     M138  ; 分度盤
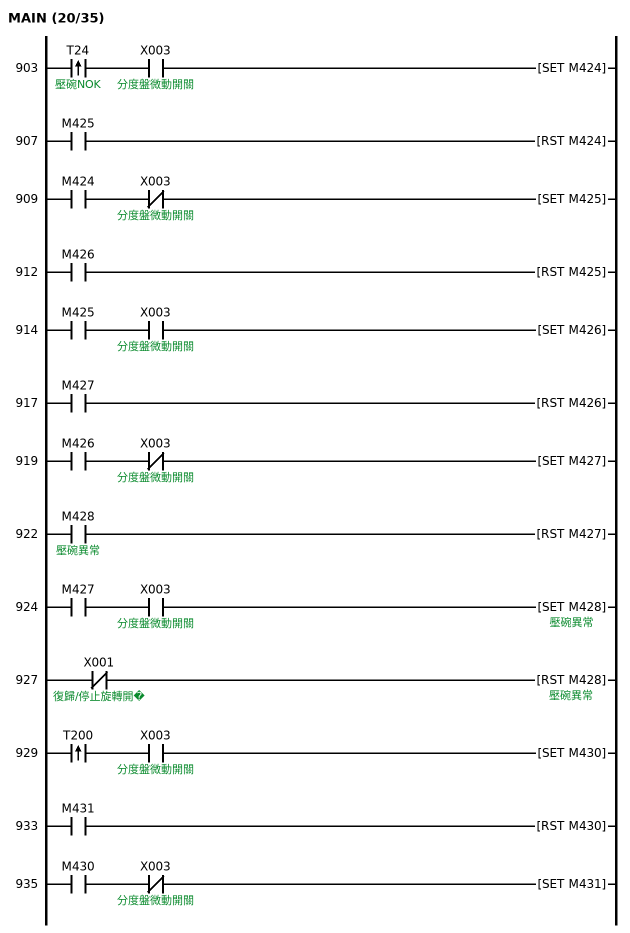
903   LDP     T24  ; 壓碗NOK
      AND     X003  ; 分度盤微動開關
      SET     M424
907   LD      M425
      RST     M424
909   LD      M424
      ANI     X003  ; 分度盤微動開關
      SET     M425
912   LD      M426
      RST     M425
914   LD      M425
      AND     X003  ; 分度盤微動開關
      SET     M426
917   LD      M427
      RST     M426
919   LD      M426
      ANI     X003  ; 分度盤微動開關
      SET     M427
922   LD      M428  ; 壓碗異常
      RST     M427
924   LD      M427
      AND     X003  ; 分度盤微動開關
      SET     M428  ; 壓碗異常
927   LDI     X001  ; 復歸/停止旋轉開�
      RST     M428  ; 壓碗異常
929   LDP     T200
      AND     X003  ; 分度盤微動開關
      SET     M430
933   LD      M431
      RST     M430
935   LD      M430
      ANI     X003  ; 分度盤微動開關
      SET     M431
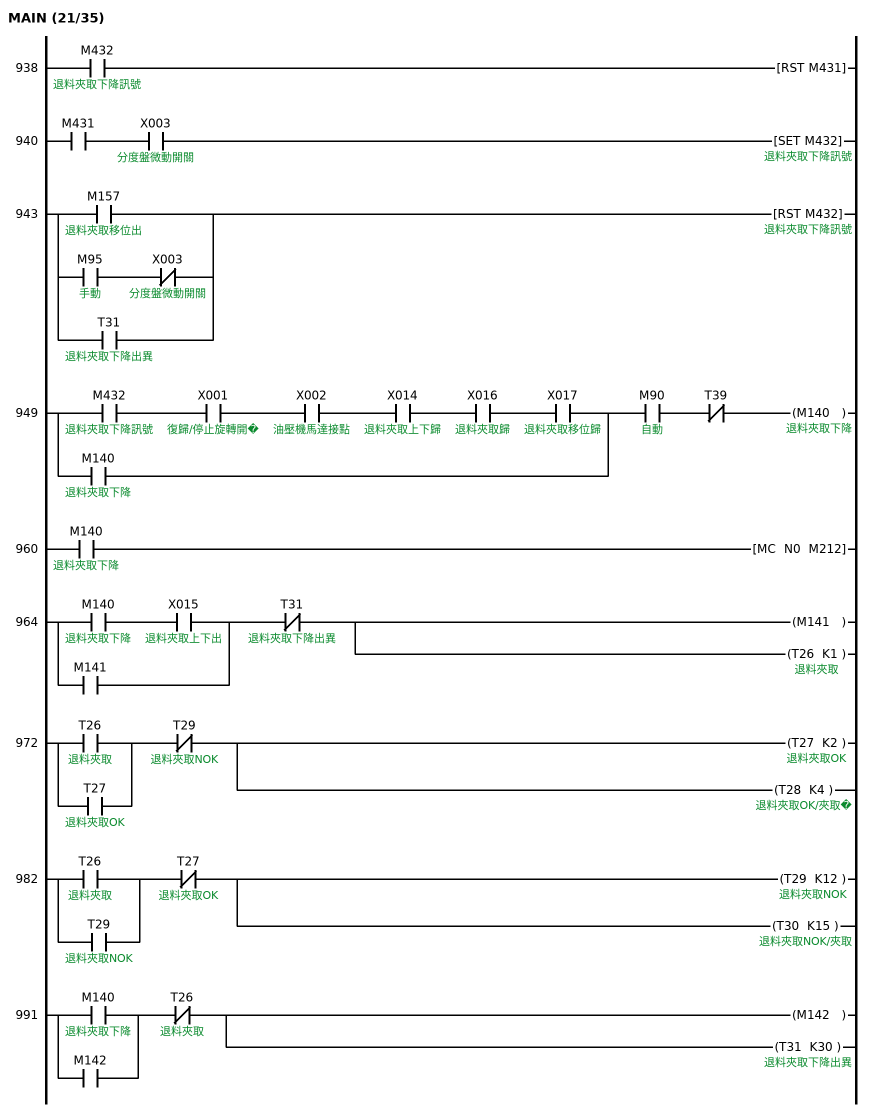
938   LD      M432  ; 退料夾取下降訊號
      RST     M431
940   LD      M431
      AND     X003  ; 分度盤微動開關
      SET     M432  ; 退料夾取下降訊號
943   LD      M157  ; 退料夾取移位出
      LD      M95  ; 手動
      ANI     X003  ; 分度盤微動開關
      ORB
      OR      T31  ; 退料夾取下降出異
      RST     M432  ; 退料夾取下降訊號
949   LD      M432  ; 退料夾取下降訊號
      AND     X001  ; 復歸/停止旋轉開�
      AND     X002  ; 油壓機馬達接點
      AND     X014  ; 退料夾取上下歸
      AND     X016  ; 退料夾取歸
      AND     X017  ; 退料夾取移位歸
      OR      M140  ; 退料夾取下降
      AND     M90  ; 自動
      ANI     T39
      OUT     M140  ; 退料夾取下降
960   LD      M140  ; 退料夾取下降
      MC      N0 M212
964   LD      M140  ; 退料夾取下降
      AND     X015  ; 退料夾取上下出
      OR      M141
      ANI     T31  ; 退料夾取下降出異
      OUT     M141
      OUT     T26 K1  ; 退料夾取
972   LD      T26  ; 退料夾取
      OR      T27  ; 退料夾取OK
      ANI     T29  ; 退料夾取NOK
      OUT     T27 K2  ; 退料夾取OK
      OUT     T28 K4  ; 退料夾取OK/夾取�
982   LD      T26  ; 退料夾取
      OR      T29  ; 退料夾取NOK
      ANI     T27  ; 退料夾取OK
      OUT     T29 K12  ; 退料夾取NOK
      OUT     T30 K15  ; 退料夾取NOK/夾取
991   LD      M140  ; 退料夾取下降
      OR      M142
      ANI     T26  ; 退料夾取
      OUT     M142
      OUT     T31 K30  ; 退料夾取下降出異
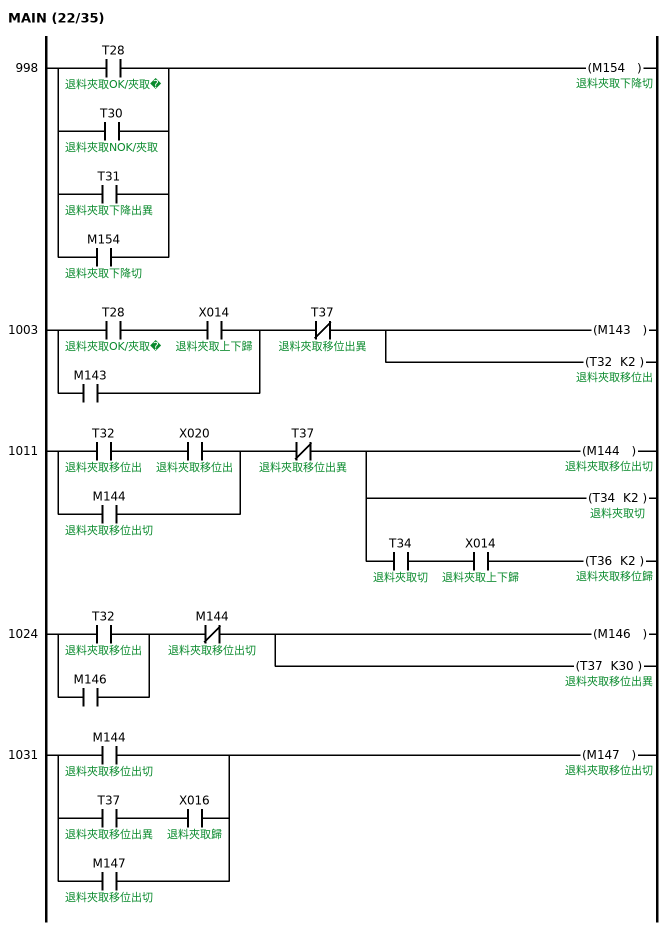
998   LD      T28  ; 退料夾取OK/夾取�
      OR      T30  ; 退料夾取NOK/夾取
      OR      T31  ; 退料夾取下降出異
      OR      M154  ; 退料夾取下降切
      OUT     M154  ; 退料夾取下降切
1003  LD      T28  ; 退料夾取OK/夾取�
      AND     X014  ; 退料夾取上下歸
      OR      M143
      ANI     T37  ; 退料夾取移位出異
      OUT     M143
      OUT     T32 K2  ; 退料夾取移位出
1011  LD      T32  ; 退料夾取移位出
      AND     X020  ; 退料夾取移位出
      OR      M144  ; 退料夾取移位出切
      ANI     T37  ; 退料夾取移位出異
      OUT     M144  ; 退料夾取移位出切
      OUT     T34 K2  ; 退料夾取切
      AND     T34  ; 退料夾取切
      AND     X014  ; 退料夾取上下歸
      OUT     T36 K2  ; 退料夾取移位歸
1024  LD      T32  ; 退料夾取移位出
      OR      M146
      ANI     M144  ; 退料夾取移位出切
      OUT     M146
      OUT     T37 K30  ; 退料夾取移位出異
1031  LD      M144  ; 退料夾取移位出切
      LD      T37  ; 退料夾取移位出異
      AND     X016  ; 退料夾取歸
      ORB
      OR      M147  ; 退料夾取移位出切
      OUT     M147  ; 退料夾取移位出切
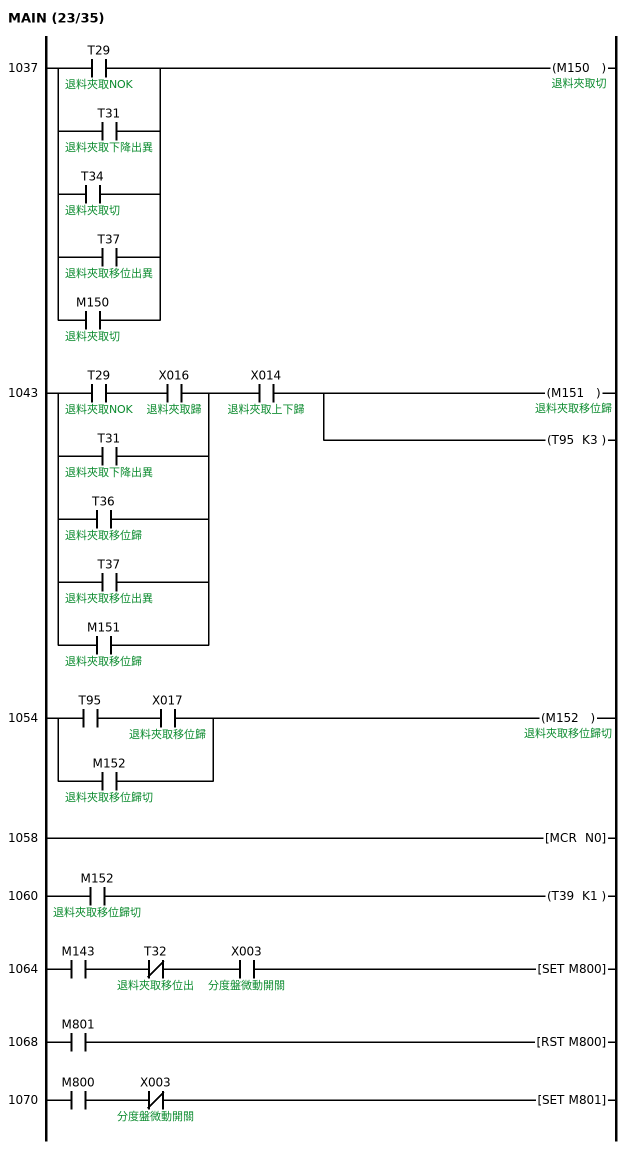
1037  LD      T29  ; 退料夾取NOK
      OR      T31  ; 退料夾取下降出異
      OR      T34  ; 退料夾取切
      OR      T37  ; 退料夾取移位出異
      OR      M150  ; 退料夾取切
      OUT     M150  ; 退料夾取切
1043  LD      T29  ; 退料夾取NOK
      AND     X016  ; 退料夾取歸
      OR      T31  ; 退料夾取下降出異
      OR      T36  ; 退料夾取移位歸
      OR      T37  ; 退料夾取移位出異
      OR      M151  ; 退料夾取移位歸
      AND     X014  ; 退料夾取上下歸
      OUT     M151  ; 退料夾取移位歸
      OUT     T95 K3
1054  LD      T95
      AND     X017  ; 退料夾取移位歸
      OR      M152  ; 退料夾取移位歸切
      OUT     M152  ; 退料夾取移位歸切
1058  MCR     N0
1060  LD      M152  ; 退料夾取移位歸切
      OUT     T39 K1
1064  LD      M143
      ANI     T32  ; 退料夾取移位出
      AND     X003  ; 分度盤微動開關
      SET     M800
1068  LD      M801
      RST     M800
1070  LD      M800
      ANI     X003  ; 分度盤微動開關
      SET     M801
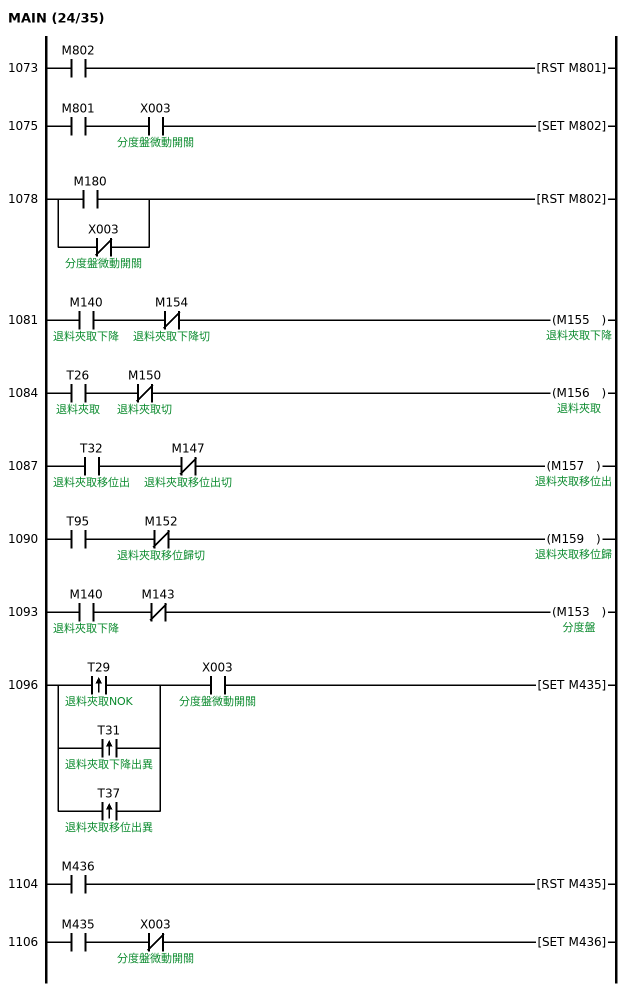
1073  LD      M802
      RST     M801
1075  LD      M801
      AND     X003  ; 分度盤微動開關
      SET     M802
1078  LD      M180
      ORI     X003  ; 分度盤微動開關
      RST     M802
1081  LD      M140  ; 退料夾取下降
      ANI     M154  ; 退料夾取下降切
      OUT     M155  ; 退料夾取下降
1084  LD      T26  ; 退料夾取
      ANI     M150  ; 退料夾取切
      OUT     M156  ; 退料夾取
1087  LD      T32  ; 退料夾取移位出
      ANI     M147  ; 退料夾取移位出切
      OUT     M157  ; 退料夾取移位出
1090  LD      T95
      ANI     M152  ; 退料夾取移位歸切
      OUT     M159  ; 退料夾取移位歸
1093  LD      M140  ; 退料夾取下降
      ANI     M143
      OUT     M153  ; 分度盤
1096  LDP     T29  ; 退料夾取NOK
      ORP     T31  ; 退料夾取下降出異
      ORP     T37  ; 退料夾取移位出異
      AND     X003  ; 分度盤微動開關
      SET     M435
1104  LD      M436
      RST     M435
1106  LD      M435
      ANI     X003  ; 分度盤微動開關
      SET     M436
